// TIA Portal V20 export
TYPE "UDT_OPCButtons"
   STRUCT
      bBlink : Bool;   // From PLC
      bClick : Bool;   // From HMI
      bEnable : Bool;   // From PLC
      bIsPressed : Bool;   // From PLC
      eColor : Int;   // From PLC
   END_STRUCT;
END_TYPE
